FUNCTION_BLOCK ILOCK_SWITCH_PROTECT (* Prioritizes the last active input with a protection dead-time before switching. *)
  (* Standard: 61499-2; Description: Copyright (c) 2023 HR Agrartechnik GmbH This program and the accompanying materials are made available under the terms of the Eclipse Public License 2.0 which is available at https://www.eclipse.org/legal/epl-2.0/ SPDX-License-Identifier: EPL-2.0 *)
  (* Version 1.0, 2026-04-19, Franz Höpfinger, HR Agrartechnik GmbH, initial API and implementation and/or initial documentation *)
  PACKAGE logiBUS::signalprocessing::interlock;
  IMPORT eclipse4diac::core::TypeHash;
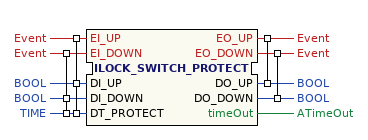
  EVENT_INPUT
    EI_UP WITH DI_UP, DT_PROTECT;
    EI_DOWN WITH DI_DOWN, DT_PROTECT;
  END_EVENT
  EVENT_OUTPUT
    EO_UP WITH DO_UP;
    EO_DOWN WITH DO_DOWN;
  END_EVENT
  VAR_INPUT
    DI_UP : BOOL; (* TRUE = forward, up, right, clockwise *)
    DI_DOWN : BOOL; (* TRUE = backward, down, left, counter-clockwise *)
    DT_PROTECT : TIME := T#50ms; (* Protection Dead-Time *)
  END_VAR
  VAR_OUTPUT
    DO_UP : BOOL; (* TRUE = forward, up, right, clockwise *)
    DO_DOWN : BOOL; (* TRUE = backward, down, left, counter-clockwise *)
  END_VAR
  PLUGS
    timeOut : iec61499::events::ATimeOut; (* Protection Timer Adapter *)
  END_PLUGS
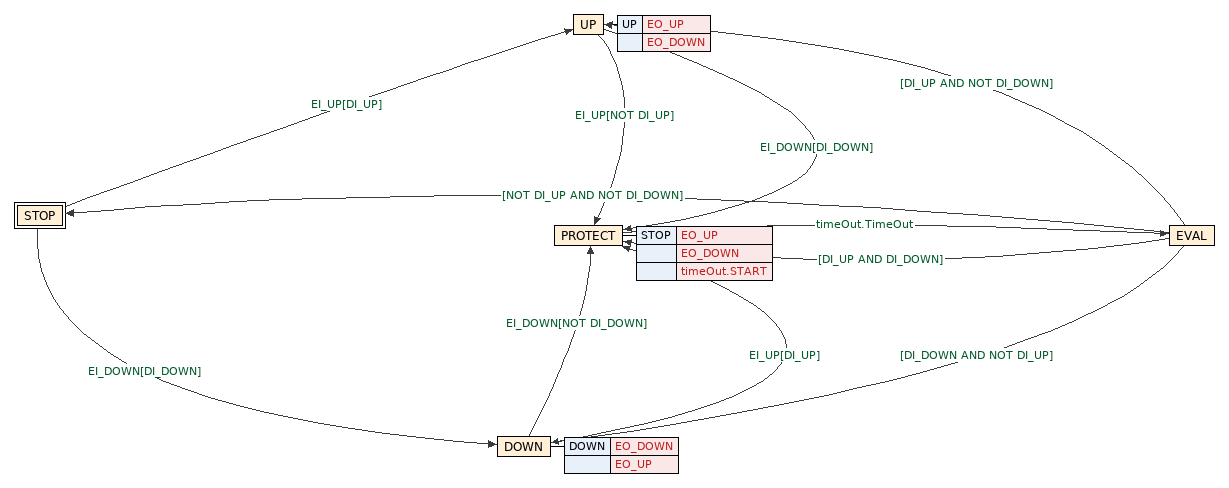
  EC_STATES
    STOP;
    UP : UP -> EO_UP, -> EO_DOWN;
    DOWN : DOWN -> EO_DOWN, -> EO_UP;
    PROTECT : STOP -> EO_UP, -> EO_DOWN, -> timeOut.START;
    EVAL;
  END_STATES
  EC_TRANSITIONS
    STOP TO UP := EI_UP[DI_UP];
    STOP TO DOWN := EI_DOWN[DI_DOWN];
    UP TO PROTECT := EI_UP[NOT DI_UP];
    UP TO PROTECT := EI_DOWN[DI_DOWN];
    DOWN TO PROTECT := EI_DOWN[NOT DI_DOWN];
    DOWN TO PROTECT := EI_UP[DI_UP];
    PROTECT TO EVAL := timeOut.TimeOut;
    EVAL TO UP := [DI_UP AND NOT DI_DOWN];
    EVAL TO DOWN := [DI_DOWN AND NOT DI_UP];
    EVAL TO STOP := [NOT DI_UP AND NOT DI_DOWN];
    EVAL TO PROTECT := [DI_UP AND DI_DOWN];
  END_TRANSITIONS
  ALGORITHM UP IN ST:
timeOut.DT := DT_PROTECT;
DO_UP := BOOL#TRUE;
DO_DOWN := BOOL#FALSE;
  END_ALGORITHM
  ALGORITHM DOWN IN ST:
timeOut.DT := DT_PROTECT;
DO_UP := BOOL#FALSE;
DO_DOWN := BOOL#TRUE;
  END_ALGORITHM
  ALGORITHM STOP IN ST:
timeOut.DT := DT_PROTECT;
DO_UP := BOOL#FALSE;
DO_DOWN := BOOL#FALSE;
  END_ALGORITHM
END_FUNCTION_BLOCK
